Fanuc KAREL source: port_RDI.kl

PROGRAM TP
%NOLOCKGROUP
VAR
 x: BOOLEAN
BEGIN
 x = RDI[3]
END TP
